DATA_BLOCK "DB"
{ S7_Optimized_Access := 'true' }
    VAR
        S_an_output: DINT;
        S_a_wire: BOOL;
        S_data: LREAL;
        avalue: DINT;
        flag: BOOL;
        measurement: LREAL;
        firstRun: BOOL;
    END_VAR
BEGIN
    firstRun := TRUE;
END_DATA_BLOCK
